KUKA KRL program: Measure.src, Measure.dat

--- Measure.src ---
&ACCESS RVP
&PARAM EDITMASK = *
DEF Measure()
   ;------------------------------------------------------------------------
   ; Measure Example Program for Roboception rc_visard/rc_cube
   ;
   ; This program demonstrates depth measurement capabilities using Roboception's
   ; Measure module. The program:
   ; 1. Configures measurement parameters (cell count, pose frame, etc.)
   ; 2. Performs depth measurements with continuous monitoring
   ; 3. Retrieves and processes measurement results including:
   ;    - Cell-wise coverage and depth statistics (min, max, mean Z values)
   ;    - Overall coverage and depth statistics across all cells
   ;    - Region of interest information and dimensions
   ; 4. Continuously loops for repeated measurements until interrupted
   ;
   ; IMPORTANT SETUP INSTRUCTIONS:
   ; 1. The service names MUST match exactly with your EKI XML configuration files
   ; 2. Modify only the parameters in this section before running the program
   ; 3. Ensure the robot is positioned to view the measurement area
   ; 4. Configure cell count parameters based on your measurement requirements
   ;
   ; HOW THE PROGRAM WORKS:
   ; - The program calls the Measure detection service which performs depth analysis
   ; - Measurement results are returned as cell-based statistics including:
   ;   a) Individual cell coverage and Z-depth statistics (min, max, mean)
   ;   b) Overall measurement statistics across all cells
   ;   c) Region of interest dimensions and positioning
   ; - The program continuously loops, performing measurements until interrupted
   ; - All measurement data is displayed via RC_SETMSG for monitoring
   ;
   ; The measurement process provides detailed depth information for quality control,
   ; object detection, and spatial analysis applications.
   ;------------------------------------------------------------------------

   DECL CHAR serviceNameDetect[64]
   DECL EKI_Status RET
   DECL E6POS flangePose

   ; Service name - same as the EKI service name
   ; TODO: Change this to the correct service name - could be "sensor_a_pipeline_1_rc_measure-measure_depth"
   serviceNameDetect[] = "rc_measure-measure_depth"

   ; Init cadmatch module and open connection to rc_cube
   $FLAG[1] = FALSE
   RC_SETMSG("Start")

   ;FOLD INI;%{PE}
      ;FOLD BASISTECH INI
         GLOBAL INTERRUPT DECL 3 WHEN $STOPMESS==TRUE DO IR_STOPM ( )
         INTERRUPT ON 3
         BAS (#INITMOV,0 )
      ;ENDFOLD (BASISTECH INI)
   ;ENDFOLD (INI)

   INTERRUPT DECL 89 WHEN $FLAG[998] DO RC_NOTIFYRECEIVED(1, 998)
   INTERRUPT ON 89

   RC_INIT(serviceNameDetect[])

   LOOP

      ; Reset vision results
      WAIT SEC 0
      ResetData()

      ; Configure detection
      ConfigureDetection(serviceNameDetect[])

      ; Perform detection
      PerformDetection(serviceNameDetect[])

      ; Error handling
      IF (RETURNCODE.VALUE < 0) THEN
         RC_SETMSG("Execution failed")
         RC_SETMSG(RETURNCODE.MSG[])
         HALT
      ENDIF

   ENDLOOP

   ; No explicit close here; PerformDetection handles connection lifecycle

END

; ---- Roboception Functions ----
;FOLD ROBOCEPTION_FUNCTIONS
   DEF ConfigureDetection(serviceNameDetect[]:IN)
      DECL CHAR serviceNameDetect[]
      DECL EKI_Status RET
      DECL E6POS flangePose

      ; Mandatory application parameters
      RET = EKI_SetString(serviceNameDetect[], "req/args/pose_frame", "external")
      RET = EKI_SetInt(serviceNameDetect[], "req/args/cell_count/@x", 1)
      RET = EKI_SetInt(serviceNameDetect[], "req/args/cell_count/@y", 1)

      ; Configure region of interest
      RET = EKI_SetInt(serviceNameDetect[], "req/args/region_of_interest_2d/@height", roi_height)
      RET = EKI_SetInt(serviceNameDetect[], "req/args/region_of_interest_2d/@offset_x", roi_offset_x)
      RET = EKI_SetInt(serviceNameDetect[], "req/args/region_of_interest_2d/@offset_y", roi_offset_Y)
      RET = EKI_SetInt(serviceNameDetect[], "req/args/region_of_interest_2d/@width", roi_width)

      flangePose = $POS_ACT_MES : INV_POS($TOOL)
      RET = EKI_SetFrame(serviceNameDetect[], "req/args/robot_pose", flangePose)
   END

   DEF PerformDetection(serviceNameDetect[]:IN)
      DECL CHAR serviceNameDetect[]
      DECL EKI_Status RET

      ; Open connection before sending request
      RC_OPENCONNECTION(serviceNameDetect[])

      ; Synchronize advance run pointer
      WAIT SEC 0

      ; Send trigger and wait for vision results
      RET = EKI_Send(serviceNameDetect[], "req")
      RC_WAITFORRESULT(1)
      RC_READRESULT(serviceNameDetect[])

      ; Close after reading results
      RC_CLOSECONNECTION(serviceNameDetect[], "req")
   END

   ;FOLD RC_SETMSG
      DEF RC_SETMSG(msg[]:IN)
         DECL CHAR msg[]
         DECL KrlMsgPar_T params[3]
         RC_SETMSG_PARAM(msg[], params[])
      END
   ;ENDFOLD (RC_SETMSG)

   ;FOLD RC_SETMSG_PARAM
      DEF RC_SETMSG_PARAM(msg[]:IN, params:OUT)
         DECL CHAR msg[]
         DECL KrlMsgPar_T params[]

         DECL KrlMsg_T name
         DECL KrlMsgOpt_T options
         DECL INT Handle, len, count
         DECL EKrlMsgType Type

         name={modul[] "rc", nr 1, msg_txt[] " "}

         Type=#notify

         len=STRLEN(msg[])
         IF len>0 THEN
            IF len>80 THEN
               len=80
            ENDIF
            FOR count=1 TO len
               name.msg_txt[count]=msg[count]
            ENDFOR
         ELSE
            name.msg_txt[]="parameter msg[] is missing"
         ENDIF

         Handle=Set_KrlMsg(Type, name, params[], options)
      END
   ;ENDFOLD (RC_SETMSG_PARAM)

   ;FOLD RC_INIT
      DEF RC_INIT(configFileName[]:IN)
         DECL CHAR configFileName[]
         DECL EKI_Status RET
         RET=EKI_INIT(configFileName[])
      END
   ;ENDFOLD (RC_INIT)

   ;FOLD RC_OPENCONNECTION
      DEF RC_OPENCONNECTION(configFileName[]:IN)
         DECL CHAR configFileName[]
         DECL EKI_Status RET
         RET=EKI_Open(configFileName[])
         EKI_CHECK(RET,#Quit)
      END
   ;ENDFOLD (RC_OPENCONNECTION)

   ;FOLD RC_CLOSECONNECTION
      DEF RC_CLOSECONNECTION(configFileName[]:IN, strPlace[]:IN)
         DECL CHAR configFileName[]
         DECL CHAR strPlace[]
         DECL EKI_Status RET
         WAIT SEC 0
         RET=EKI_Close(configFileName[])
         RET=EKI_ClearBuffer(configFileName[], strPlace[])
      END
   ;ENDFOLD (RC_CLOSECONNECTION)

   ;FOLD RC_WAITFORRESULT
      DEF RC_WAITFORRESULT(WaitFlag:IN)
         DECL INT WaitFlag

         WAIT FOR $FLAG[WaitFlag] OR NOT $FLAG[RCEkiAliveFlagNo]

         ;Eki-connection has been closed

         IF(NOT $FLAG[RCEkiAliveFlagNo]) THEN
            RC_SETMSG("EKI connection lost")
         ENDIF

         $FLAG[WaitFlag] = FALSE
         WAIT SEC 0
      END
   ;ENDFOLD (RC_WAITFORRESULT)

   ;FOLD RC_NOTIFYRECEIVED
      DEF RC_NOTIFYRECEIVED(WAITFLAG:IN, EOFRESULFLAG:IN)
         DECL INT WAITFLAG
         DECL INT EOFRESULFLAG
         $FLAG[EOFRESULFLAG]=FALSE
         $FLAG[WAITFLAG]=TRUE
      END
   ;ENDFOLD (RC_NOTIFYRECEIVED)

   ;FOLD RC_READRESULT
      DEF RC_READRESULT(configFileName[]:IN)
         DECL CHAR configFileName[]
         DECL RETURNCODE_T RESULT
         DECL EKI_STATUS RET
         DECL KrlMsgPar_T par[3]

         RESULT={VALUE 0, MSG[] "0"}

         ;Receive error codes
         RET = EKI_GetInt(configFileName[], "res/return_code/@value", RESULT.VALUE)
         RET = EKI_GetString(configFileName[], "res/return_code/@message", RESULT.MSG[])
         RETURNCODE = RESULT

         ; Display error message immediately if there is one
         IF (RESULT.VALUE < 0) THEN
            RC_SETMSG("API Error")
            RC_SETMSG(RESULT.MSG[])
         ENDIF


         ;Receive data
         RET = EKI_GetInt(configFileName[], "res/cell_count/@x", cell_count_x)
         RET = EKI_GetInt(configFileName[], "res/cell_count/@y", cell_count_y)

         RET = EKI_GetReal(configFileName[], "res/cells/le/coverage", cells_le_coverage)
         RET = EKI_GetReal(configFileName[], "res/cells/le/max_z/@x", cells_le_max_z_x)
         RET = EKI_GetReal(configFileName[], "res/cells/le/max_z/@y", cells_le_max_z_y)
         RET = EKI_GetReal(configFileName[], "res/cells/le/max_z/@z", cells_le_max_z_z)
         RET = EKI_GetReal(configFileName[], "res/cells/le/mean_z/@x", cells_le_mean_z_x)
         RET = EKI_GetReal(configFileName[], "res/cells/le/mean_z/@y", cells_le_mean_z_y)
         RET = EKI_GetReal(configFileName[], "res/cells/le/mean_z/@z", cells_le_mean_z_z)
         RET = EKI_GetReal(configFileName[], "res/cells/le/min_z/@x", cells_le_min_z_x)
         RET = EKI_GetReal(configFileName[], "res/cells/le/min_z/@y", cells_le_min_z_y)
         RET = EKI_GetReal(configFileName[], "res/cells/le/min_z/@z", cells_le_min_z_z)

         RET = EKI_GetReal(configFileName[], "res/overall/@coverage", cells_overall_coverage)
         RET = EKI_GetReal(configFileName[], "res/overall/max_z/@x", cells_overall_max_z_x)
         RET = EKI_GetReal(configFileName[], "res/overall/max_z/@y", cells_overall_max_z_y)
         RET = EKI_GetReal(configFileName[], "res/overall/max_z/@z", cells_overall_max_z_z)
         RET = EKI_GetReal(configFileName[], "res/overall/mean_z/@x", cells_overall_mean_z_x)
         RET = EKI_GetReal(configFileName[], "res/overall/mean_z/@y", cells_overall_mean_z_y)
         RET = EKI_GetReal(configFileName[], "res/overall/mean_z/@z", cells_overall_mean_z_z)
         RET = EKI_GetReal(configFileName[], "res/overall/min_z/@x", cells_overall_min_z_x)
         RET = EKI_GetReal(configFileName[], "res/overall/min_z/@y", cells_overall_min_z_y)
         RET = EKI_GetReal(configFileName[], "res/overall/min_z/@z", cells_overall_min_z_z)

         RET = EKI_ClearBuffer(configFileName[], "res")

         ; Print overall mean Z measurement results on robot

         par[1] = {par_type #value, par_REAL 0}
         par[1].par_REAL = cells_overall_mean_z_x
         par[2] = {par_type #value, par_REAL 0}
         par[2].par_REAL = cells_overall_mean_z_y
         par[3] = {par_type #value, par_REAL 0}
         par[3].par_REAL = cells_overall_mean_z_z
         RC_SETMSG_PARAM("Overall Mean Z: X=%1 Y=%2 Z=%3", par[])
      END

   ;ENDFOLD (RC_READRESULT)

   ;FOLD (ResetData)
      DEF ResetData()
         cell_count_x = 0
         cell_count_y = 0
      END
   ;ENDFOLD (ResetData)
;ENDFOLD (ROBOCEPTION_FUNCTIONS)

--- Measure.dat ---
&ACCESS RVP
&PARAM EDITMASK = *
DEFDAT Measure

   ;FOLD EXTERNAL DECLARATIONS;%{PE}%MKUKATPBASIS,%CEXT,%VCOMMON,%P
   ;FOLD BASISTECH EXT;%{PE}%MKUKATPBASIS,%CEXT,%VEXT,%P
   EXT BAS (BAS_COMMAND :IN,REAL :IN )
   DECL INT SUCCESS
   ;ENDFOLD (BASISTECH EXT)

   ;FOLD USER EXT;%{E}%MKUKATPUSER,%CEXT,%VEXT,%P
   STRUC RETURNCODE_T INT VALUE,CHAR MSG[512]
   DECL RETURNCODE_T RETURNCODE
   DECL INT RCEkiAliveFlagNo=997
   ;ENDFOLD (USER EXT)
   ;ENDFOLD (EXTERNAL DECLARATIONS)

   ;FOLD MEASUREMENT DATA
   DECL CHAR pose_frame[256]
   pose_frame[]="external'H00''H00''H00''H00''H00''H00''H00''H00''H00''H00''H00''H00''H00''H00''H00''H00''H00''H00''H00''H00''H00''H00''H00''H00''H00''H00''H00''H00''H00''H00''H00''H00''H00''H00''H00''H00''H00''H00''H00''H00''H00''H00''H00''H00''H00''H00''H00''H00''H00''H00''H00''H00''H00''H00''H00''H00''H00''H00''H00''H00''H00''H00''H00''H00''H00''H00''H00''H00''H00''H00''H00''H00''H00''H00''H00''H00''H00''H00''H00''H00''H00''H00''H00''H00''H00''H00''H00''H00''H00''H00''H00''H00''H00''H00''H00''H00''H00''H00''H00''H00''H00''H00''H00''H00''H00''H00''H00''H00''H00''H00''H00''H00''H00''H00''H00''H00''H00''H00''H00''H00''H00''H00''H00''H00''H00''H00''H00''H00''H00''H00''H00''H00''H00''H00''H00''H00''H00''H00''H00''H00''H00''H00''H00''H00''H00''H00''H00''H00''H00''H00''H00''H00''H00''H00''H00''H00''H00''H00''H00''H00''H00''H00''H00''H00''H00''H00''H00''H00''H00''H00''H00''H00''H00''H00''H00''H00''H00''H00''H00''H00''H00''H00''H00''H00''H00''H00''H00''H00''H00''H00''H00''H00''H00''H00''H00''H00''H00''H00''H00''H00''H00''H00''H00''H00''H00''H00''H00''H00''H00''H00''H00''H00''H00''H00''H00''H00''H00''H00''H00''H00''H00''H00''H00''H00''H00''H00''H00''H00''H00''H00''H00''H00''H00''H00''H00''H00''H00''H00''H00''H00''H00''H00''H00''H00''H00''H00''H00''H00'"

   DECL INT cell_count_x=1
   DECL INT cell_count_y=1

   DECL REAL cells_le_coverage=0.0
   DECL REAL cells_le_max_z_x=0.0
   DECL REAL cells_le_max_z_y=0.0
   DECL REAL cells_le_max_z_z=0.0
   DECL REAL cells_le_mean_z_x=0.0
   DECL REAL cells_le_mean_z_y=0.0
   DECL REAL cells_le_mean_z_z=0.0
   DECL REAL cells_le_min_z_x=0.0
   DECL REAL cells_le_min_z_y=0.0
   DECL REAL cells_le_min_z_z=0.0

   DECL REAL cells_overall_coverage=0.0
   DECL REAL cells_overall_max_z_x=0.0
   DECL REAL cells_overall_max_z_y=0.0
   DECL REAL cells_overall_max_z_z=0.0
   DECL REAL cells_overall_mean_z_x=0.0
   DECL REAL cells_overall_mean_z_y=0.0
   DECL REAL cells_overall_mean_z_z=0.0
   DECL REAL cells_overall_min_z_x=0.0
   DECL REAL cells_overall_min_z_y=0.0
   DECL REAL cells_overall_min_z_z=0.0
   ;ENDFOLD (MEASUREMENT DATA)

   ;FOLD ROI
   DECL INT roi_height=960
   DECL INT roi_offset_x=0
   DECL INT roi_offset_Y=0
   DECL INT roi_width=1280
   ;ENDFOLD (ROI)

   ; Movement data
   DECL LDAT lDatDefault={VEL 2.00000,ACC 20.0000,APO_DIST 10.0000,APO_FAC 50.0000,AXIS_VEL 100.000,AXIS_ACC 100.000,ORI_TYP #VAR,CIRC_TYP #BASE,JERK_FAC 50.0000,GEAR_JERK 100.000,EXAX_IGN 0,CB {AUX_PT {ORI #CONSIDER,E1 #CONSIDER,E2 #CONSIDER,E3 #CONSIDER,E4 #CONSIDER,E5 #CONSIDER,E6 #CONSIDER},TARGET_PT {ORI #INTERPOLATE,E1 #INTERPOLATE,E2 #INTERPOLATE,E3 #INTERPOLATE,E4 #INTERPOLATE,E5 #INTERPOLATE,E6 #INTERPOLATE}}}
   DECL FDAT fDatDefault={TOOL_NO 4,BASE_NO 0,IPO_FRAME #BASE,POINT2[] " "}
   DECL PDAT pDatDefault={VEL 10.0000,ACC 20.0000,APO_DIST 10.0000,APO_MODE #CDIS,GEAR_JERK 100.000,EXAX_IGN 0}

ENDDAT
